(* IEC 61131-3 sources: Fosela-House-/control/free_smart, 5 files *)

(* ---- GVL_Smart.st ---- *)
(* ============================================================
   GVL_Smart.st
   Variables globales del controlador solar (controlador esclavo Modbus).
   Subsistema solar — Fusela House
   ============================================================ *)

VAR_GLOBAL

    (* ---- Entradas analógicas (sondas NTC/Pt1000) ---- *)
    TT1             : REAL;     (* AI1 — temperatura salida colector [°C] *)
    TT2             : REAL;     (* AI2 — D1 fondo [°C] *)
    TT3             : REAL;     (* AI3 — D1 cabeza [°C] *)

    (* ---- Salidas analógicas ---- *)
    AO_P1_speed     : REAL;     (* AO 0-10V → convertidor PWM → bomba solar modulante [V] *)

    (* ---- Salidas digitales (relés) ---- *)
    DO_V3V_SOL      : BOOL;     (* Relé 1: FALSE=serp.inf D1 (ACS), TRUE=serp.sup D1 (piscina) *)
    DO_PERS_SOL     : BOOL;     (* Relé 2: FALSE=abiertas, TRUE=cerradas *)
    DO_P2           : BOOL;     (* Relé 3: bomba mini bucle intermedio *)
    DO_ALM_SOLAR    : BOOL;     (* Relé 4: alarma local solar *)

    (* ---- Datos calculados para publicación Modbus ---- *)
    DT_solar        : REAL;     (* ΔT medido TT1 - TT2 [K] *)
    vel_P1_permil   : UINT;     (* Velocidad P1 en ‰ (0-1000) *)

    (* ---- Setpoints recibidos del FRE via Modbus (registros 200-203) ---- *)
    SP_DT_solar     : REAL := 8.0;          (* ΔT objetivo P1 [K] *)
    modo_solar      : E_Solar_Mode := SOLAR_AUTO;
    orden_persianas : BOOL := FALSE;        (* FALSE=auto, TRUE=forzar cierre *)
    SP_TT3_piscina  : REAL := 75.0;         (* TT3 mínimo para desvío a piscina [°C] *)

    (* ---- Alarmas ---- *)
    ALM_TT1_HIGH    : BOOL;
    ALM_TT2_HIGH    : BOOL;
    alarma_solar_code : UINT;   (* 0=OK, 1=TT1 alta, 2=TT2 alta, 3=ambas *)

END_VAR

(* ---- FB_SolarPump.st ---- *)
(* ============================================================
   FB_SolarPump.st
   Control de la bomba solar P1 (modulante via convertidor 0-10V→PWM).
   - Lazo PI discreto de ΔT constante
   - Tiempos mínimos anti-ciclado
   - Modos: AUTO, OFF, FORZADO
   ============================================================ *)

FUNCTION_BLOCK FB_SolarPump

VAR_INPUT
    TT1             : REAL;     (* Temperatura colector [°C] *)
    TT2             : REAL;     (* D1 fondo [°C] *)
    SP_DT           : REAL;     (* ΔT objetivo [K] *)
    mode            : E_Solar_Mode;
    fault           : BOOL := FALSE;
END_VAR

VAR_OUTPUT
    pump_run        : BOOL;     (* Orden de marcha a FB_Pump *)
    speed_pct       : REAL;     (* Velocidad [0-100 %] → mapear a 0-10V *)
    DT_measured     : REAL;     (* ΔT actual TT1-TT2 *)
    state_desc      : STRING;   (* Descripción estado para diagnóstico *)
END_VAR

VAR
    pi              : FB_PI_Controller;
    pump            : FB_Pump;
    DT_current      : REAL;
    pi_enabled      : BOOL;
END_VAR

(* --- Implementación --- *)

DT_current  := TT1 - TT2;
DT_measured := DT_current;

(* Decidir si P1 debe marchar *)
CASE mode OF

    SOLAR_AUTO:
        (* Arranque diferencial: DT > C_SOLAR_DT_START *)
        (* Parada diferencial:   DT < C_SOLAR_DT_STOP  *)
        (* (la histéresis la gestiona FB_Pump via min_on/min_off) *)
        pump_run := (DT_current > C_SOLAR_DT_START) OR
                    (pump.running AND DT_current > C_SOLAR_DT_STOP);
        pi_enabled := pump_run;
        state_desc := 'AUTO';

    SOLAR_FORCE_ACS, SOLAR_FORCE_POOL:
        pump_run   := TRUE;
        pi_enabled := TRUE;
        state_desc := 'FORZADO';

    SOLAR_OFF:
        pump_run   := FALSE;
        pi_enabled := FALSE;
        state_desc := 'OFF';

    ELSE
        pump_run   := FALSE;
        pi_enabled := FALSE;
        state_desc := 'DESCONOCIDO';
END_CASE

IF fault THEN
    pump_run   := FALSE;
    pi_enabled := FALSE;
    state_desc := 'FALLO';
END_IF

(* Lazo PI: error = ΔT_objetivo - ΔT_medido
   Si DT_current > SP_DT → error negativo → bajar caudal (bajar velocidad)
   Si DT_current < SP_DT → error positivo → subir caudal  *)
pi(
    measured    := DT_current,
    setpoint    := SP_DT,
    Kp          := 0.5,
    Ki          := 0.08,
    out_min     := 10.0,    (* Mínimo 10% para evitar cavitación a velocidad cero *)
    out_max     := 100.0,
    dt_seconds  := 1.0,
    enabled     := pi_enabled,
    reset       := NOT pump_run
);

(* Gestor de bomba (anti-ciclado) *)
pump(
    cmd_run      := pump_run,
    fault        := fault,
    min_on_time  := C_SOLAR_MIN_ON_TIME,
    min_off_time := C_SOLAR_MIN_OFF_TIME
);

(* Velocidad: si la bomba no corre → 0; si corre → salida PI *)
IF pump.running THEN
    speed_pct := pi.output;
ELSE
    speed_pct := 0.0;
END_IF

END_FUNCTION_BLOCK

(* ---- FB_SolarValves.st ---- *)
(* ============================================================
   FB_SolarValves.st
   Gestión de V3V_SOL, P2 (mini bucle) y PERS_SOL (persianas).

   Reglas de arbitraje V3V_SOL:
   - Por defecto: posición A (ACS) — serp.inf D1
   - Desvío a piscina (pos. B) si:
       * modo = SOLAR_FORCE_POOL, O
       * modo = SOLAR_AUTO AND TT3 >= SP_TT3_pool AND pool_demand=TRUE
   - Persianas: cierran si TT2 >= P17_SolarOverheatShutterClose o forzado externo
   - P2 (mini bucle): marcha si V3V_SOL está en posición B (piscina)
   ============================================================ *)

FUNCTION_BLOCK FB_SolarValves

VAR_INPUT
    TT2             : REAL;         (* D1 fondo [°C] *)
    TT3             : REAL;         (* D1 cabeza [°C] *)
    SP_TT3_pool     : REAL;         (* Umbral TT3 para desvío a piscina *)
    pool_demand     : BOOL;         (* TRUE = piscina necesita calor *)
    mode            : E_Solar_Mode;
    force_shutters  : BOOL;         (* TRUE = forzar cierre persianas (del FRE) *)
    pump_running    : BOOL;         (* P1 en marcha *)
    fault           : BOOL := FALSE;
END_VAR

VAR_OUTPUT
    cmd_V3V_SOL_pool : BOOL;        (* TRUE = posición B (piscina) *)
    cmd_P2_run       : BOOL;        (* TRUE = arrancar P2 *)
    cmd_shutters_close : BOOL;      (* TRUE = cerrar persianas *)
    dissipation_active : BOOL;      (* TRUE = disipación activa *)
END_VAR

VAR
    valve_sol       : FB_Valve3Way;
    pump_P2         : FB_Pump;
    want_pool       : BOOL;
    want_dissipate  : BOOL;
END_VAR

(* --- Lógica de desvío a piscina --- *)
CASE mode OF
    SOLAR_FORCE_POOL:
        want_pool := TRUE;

    SOLAR_AUTO:
        want_pool := (TT3 >= SP_TT3_pool) AND pool_demand AND pump_running;

    SOLAR_FORCE_DHW, SOLAR_OFF:
        want_pool := FALSE;
END_CASE

IF fault THEN
    want_pool := FALSE;
END_IF

(* --- V3V_SOL --- *)
valve_sol(
    cmd_pos_B   := want_pool,
    enabled     := NOT fault,
    travel_time := K_VALVE_TRAVEL
);
cmd_V3V_SOL_pool := valve_sol.DO_valve;

(* --- P2: solo corre si V3V_SOL está en posición piscina Y no en maniobra --- *)
cmd_P2_run := valve_sol.DO_valve AND
              NOT valve_sol.in_transit AND
              pump_running AND
              NOT fault;

(* --- Persianas: cierre por disipación o forzado externo --- *)
want_dissipate := (TT2 >= P17_SolarOverheatShutterClose);
dissipation_active := want_dissipate;

cmd_shutters_close := want_dissipate OR force_shutters OR fault;

END_FUNCTION_BLOCK

(* ---- MB_Slave_Map.st ---- *)
(* ============================================================
   MB_Slave_Map.st
   Mapa de registros Modbus del controlador solar (esclavo Modbus dir. 1).

   CONFIGURACIÓN EN FREE STUDIO PLUS:
   En Device → Modbus RTU Slave → Memory Mapping, mapear:
     - Holding Registers 100-108: área de lectura (FRE lee)
     - Holding Registers 200-203: área de escritura (FRE escribe)

   Este PROGRAM prepara los valores en las variables globales
   que el driver Modbus publicará automáticamente.
   Se llama en cada ciclo del PLC_PRG.

   Encoding temperatura: REAL → INT multiplicando ×10
     Ejemplo: 42.5 °C → 425 (INT)
     Límite: ±3276.7 °C — suficiente para todas las sondas
   ============================================================ *)

PROGRAM MB_Slave_Map

(* ---- Variables publicadas como Holding Registers (FRE lee) ---- *)
VAR_GLOBAL

    (* Reg 100 *) MB_OUT_TT1          : INT;  (* TT1 ×10 *)
    (* Reg 101 *) MB_OUT_TT2          : INT;  (* TT2 ×10 *)
    (* Reg 102 *) MB_OUT_TT3          : INT;  (* TT3 ×10 *)
    (* Reg 103 *) MB_OUT_VEL_P1       : UINT; (* velocidad P1 ‰ 0-1000 *)
    (* Reg 104 *) MB_OUT_V3VSOL_POS   : UINT; (* 0=ACS, 1=piscina *)
    (* Reg 105 *) MB_OUT_PERS_CLOSED  : UINT; (* 0=abiertas, 1=cerradas *)
    (* Reg 106 *) MB_OUT_P2_RUNNING   : UINT; (* 0=parada, 1=marcha *)
    (* Reg 107 *) MB_OUT_ALM_CODE     : UINT; (* 0=OK, 1=TT1, 2=TT2, 3=ambas *)
    (* Reg 108 *) MB_OUT_DT_SOLAR     : INT;  (* ΔT medido ×10 *)

END_VAR

(* ---- Setpoints recibidos (FRE escribe en estos registros) ---- *)
VAR_GLOBAL

    (* Reg 200 *) MB_IN_SP_DT         : UINT := 80;  (* ΔT objetivo ×10 → 8.0 K *)
    (* Reg 201 *) MB_IN_MODO_SOLAR    : UINT := 0;   (* E_Solar_Mode *)
    (* Reg 202 *) MB_IN_ORD_PERS      : UINT := 0;   (* 0=auto, 1=forzar cierre *)
    (* Reg 203 *) MB_IN_SP_TT3_POOL   : UINT := 750; (* TT3 umbral ×10 → 75.0°C *)
    (* Reg 204 *) MB_IN_POOL_DEMAND   : UINT := 0;   (* 0=no demanda, 1=piscina pide calor *)

END_VAR

VAR
    (* Conversiones de entrada *)
    sp_dt_real      : REAL;
    sp_tt3_real     : REAL;
END_VAR

(* ----------------------------------------------------------------
   Actualizar registros de salida (cada ciclo)
   ---------------------------------------------------------------- *)

MB_OUT_TT1        := REAL_TO_INT(TT1 * MB_TEMP_SCALE);
MB_OUT_TT2        := REAL_TO_INT(TT2 * MB_TEMP_SCALE);
MB_OUT_TT3        := REAL_TO_INT(TT3 * MB_TEMP_SCALE);
MB_OUT_VEL_P1     := REAL_TO_UINT(vel_P1_permil);
MB_OUT_V3VSOL_POS := UINT#0;
IF DO_V3V_SOL THEN MB_OUT_V3VSOL_POS := UINT#1; END_IF
MB_OUT_PERS_CLOSED:= UINT#0;
IF DO_PERS_SOL THEN MB_OUT_PERS_CLOSED := UINT#1; END_IF
MB_OUT_P2_RUNNING := UINT#0;
IF DO_P2 THEN MB_OUT_P2_RUNNING := UINT#1; END_IF
MB_OUT_ALM_CODE   := alarma_solar_code;
MB_OUT_DT_SOLAR   := REAL_TO_INT(DT_solar * MB_TEMP_SCALE);

(* ----------------------------------------------------------------
   Decodificar registros de entrada recibidos del FRE
   ---------------------------------------------------------------- *)

sp_dt_real    := UINT_TO_REAL(MB_IN_SP_DT) / MB_TEMP_SCALE;
sp_tt3_real   := UINT_TO_REAL(MB_IN_SP_TT3_POOL) / MB_TEMP_SCALE;

(* Actualizar GVL con valores recibidos *)
IF sp_dt_real >= 3.0 AND sp_dt_real <= 20.0 THEN
    SP_DT_solar := sp_dt_real;
END_IF
IF sp_tt3_real >= 50.0 AND sp_tt3_real <= 90.0 THEN
    SP_TT3_piscina := sp_tt3_real;
END_IF

modo_solar        := INT_TO_E_Solar_Mode(UINT_TO_INT(MB_IN_MODO_SOLAR));
orden_persianas   := (MB_IN_ORD_PERS = UINT#1);
pool_demand_ext   := (MB_IN_POOL_DEMAND = UINT#1);

END_PROGRAM

(* ---- PLC_PRG_Smart.st ---- *)
(* ============================================================
   PLC_PRG_Smart.st
   Programa principal del controlador solar (controlador esclavo Modbus).
   Task cíclica: 1000 ms (térmica, no requiere ciclos cortos).

   MAPEO HARDWARE (configurar en Device → I/O en FREE Studio):
     AI1 → TT1  (NTC o Pt1000, rango -20..+150 °C)
     AI2 → TT2
     AI3 → TT3
     AO1 0-10V → DO_AO_P1 (mapear a GVL AO_P1_speed)
     Relay 1    → DO_V3V_SOL
     Relay 2    → DO_PERS_SOL
     Relay 3    → DO_P2
     Relay 4    → DO_ALM_SOLAR
   ============================================================ *)

PROGRAM PLC_PRG

VAR
    (* Instancias de function blocks *)
    solar_pump      : FB_SolarPump;
    solar_valves    : FB_SolarValves;
    alm_TT1_high    : FB_Alarm;
    alm_TT2_high    : FB_Alarm;

    (* Conversión velocidad PWM *)
    speed_volt      : REAL;     (* 0-10V para la salida analógica *)

    (* Pool demand externa recibida por Modbus *)
    pool_demand_ext : BOOL := FALSE;
END_VAR

(* ============================================================
   1. ACTUALIZAR SETPOINTS DESDE MODBUS
      (MB_Slave_Map escribe en GVL_Smart: SP_DT_solar,
       SP_TT3_piscina, modo_solar, orden_persianas)
   ============================================================ *)
MB_Slave_Map();

(* ============================================================
   2. CONTROL DE BOMBA SOLAR P1
   ============================================================ *)
solar_pump(
    TT1     := TT1,
    TT2     := TT2,
    SP_DT   := SP_DT_solar,
    mode    := modo_solar,
    fault   := ALM_TT1_HIGH
);

(* Mapear velocidad % → 0-10V para AO → convertidor 0-10V→PWM → bomba solar modulante *)
speed_volt      := solar_pump.speed_pct / 10.0;   (* 0-100% → 0.0-10.0 V *)
AO_P1_speed     := speed_volt;

(* Publicar velocidad en ‰ para Modbus *)
vel_P1_permil   := REAL_TO_UINT(solar_pump.speed_pct * 10.0);
DT_solar        := solar_pump.DT_measured;

(* ============================================================
   3. CONTROL DE VÁLVULAS Y PERSIANAS
   ============================================================ *)
solar_valves(
    TT2             := TT2,
    TT3             := TT3,
    SP_TT3_pool     := SP_TT3_piscina,
    pool_demand     := pool_demand_ext,
    mode            := modo_solar,
    force_shutters  := orden_persianas,
    pump_running    := solar_pump.pump_run,
    fault           := ALM_TT1_HIGH
);

DO_V3V_SOL  := solar_valves.cmd_V3V_SOL_pool;
DO_PERS_SOL := solar_valves.cmd_shutters_close;
DO_P2       := solar_valves.cmd_P2_run;

(* ============================================================
   4. ALARMAS
   ============================================================ *)

(* Alarma TT1 alta — sobretemperatura colector *)
alm_TT1_high(
    condition   := (TT1 > C_ALM_TT1_MAX),
    reset_cmd   := FALSE,      (* Rearme automático cuando T baja *)
    filter_time := C_ALM_FILTER_TIME,
    latch       := FALSE,
    enabled     := TRUE
);
ALM_TT1_HIGH := alm_TT1_high.active;

(* Alarma TT2 alta — sobretemperatura D1 *)
alm_TT2_high(
    condition   := (TT2 > C_ALM_TT2_MAX),
    reset_cmd   := FALSE,
    filter_time := C_ALM_FILTER_TIME,
    latch       := FALSE,
    enabled     := TRUE
);
ALM_TT2_HIGH := alm_TT2_high.active;

(* Código de alarma compuesto *)
alarma_solar_code := UINT#0;
IF ALM_TT1_HIGH AND NOT ALM_TT2_HIGH THEN
    alarma_solar_code := UINT#1;
ELSIF NOT ALM_TT1_HIGH AND ALM_TT2_HIGH THEN
    alarma_solar_code := UINT#2;
ELSIF ALM_TT1_HIGH AND ALM_TT2_HIGH THEN
    alarma_solar_code := UINT#3;
END_IF

(* Relé de alarma local *)
DO_ALM_SOLAR := ALM_TT1_HIGH OR ALM_TT2_HIGH;

(* ============================================================
   5. PUBLICAR REGISTROS MODBUS (ya llamado al inicio, se repite
      para asegurar que las salidas calculadas quedan en los
      registros antes del siguiente polling del maestro)
   ============================================================ *)
MB_Slave_Map();

END_PROGRAM
